(* Logix 5000 project; controller reports 1756-L63 rev 20.11; software revision 20.04; part 52 of 52 *)
(* tags used below, declared in another part *)
   AIT501do : PRANALOG;   // Aeration tank 1 DO
   AIT501ph : PRANALOG;   // Aeration tank 1 pH
   AIT502do : PRANALOG;   // Aeration tank 2 DO
   AIT502ph : PRANALOG;   // Aeration tank 2 pH
   B301 : MOTOR;   // Equalization blower 1
   B302 : MOTOR;   // Equalization blower 2
   B303 : MOTOR;   // Equalization blower 3
   B501 : MOTOR;   // Aeration tank 1 blower 1
   B502 : MOTOR;   // Aeration tank standby blower
   B503 : MOTOR;   // Aeration tank 2 blower 1
   B601 : MOTOR;   // Membrane tank 1 blower
   B602 : MOTOR;   // Membrane tank 2 blower
   B603 : MOTOR;   // Membrane tank 3 blower
   B604 : MOTOR;   // Membrane tank 4 blower
   B901 : MOTOR;   // Digester blower 1
   B902 : MOTOR;   // Digester blower 2
   DIESEL : MOTOR;   // Diesel generator
   FIT201 : PRANALOG;   // Plant influent flow to screens
   FIT701 : PRANALOG;   // Membrane tank 1 permeate flow
   FIT702 : PRANALOG;   // Membrane tank 2 permeate flow
   FIT703 : PRANALOG;   // Membrane tank 3 permeate flow
   FIT704 : PRANALOG;   // Membrane tank 4 permeate flow
   FIT801 : PRANALOG;   // CIP flow
   FIT901 : PRANALOG;   // Membrane tanks 1 & 2 WAS flow
   FIT902 : PRANALOG;   // Membrane tanks 3 & 4 WAS flow
   FunctionBlock_Cycle_Time : REAL;   // Main Task Cycle Time in mseconds
   GT7951 : PRANALOG;   // Screening area H2S monitor
   LIT302 : PRANALOG;   // Equalization tank 302 Level
   LIT501 : PRANALOG;   // Aeration tank 1 Level
   LIT502 : PRANALOG;   // Aeration tank 2 Level
   LIT6101 : PRANALOG;   // Coagulant tank 6101 level
   LIT6102 : PRANALOG;   // Caustic tank 6102 Leve
   P301 : MOTOR;   // Equalization pump 1
   P302 : MOTOR;   // Equalization pump 2
   P303 : MOTOR;   // Equalization pump 3
   P501 : MOTOR;   // Membrane tank 1 mixed liquor pump
   P502 : MOTOR;   // Membrane tank 2 mixed liquor pump
   P503 : MOTOR;   // Membrane tank 3 mixed liquor pump
   P504 : MOTOR;   // Membrane tank 4 mixed liquor pump
   P7011 : MOTOR;   // Membrane tank 1 permeate pump 1
   P7012 : MOTOR;   // Membrane tank 1 permeate pump 2
   P7021 : MOTOR;   // Membrane tank 2 permeate pump 1
   P7022 : MOTOR;   // Membrane tank 2 permeate pump 2
   P7031 : MOTOR;   // Membrane tank 3 permeate pump 1
   P7032 : MOTOR;   // Membrane tank 3 permeate pump 2
   P7041 : MOTOR;   // Membrane tank 4 permeate pump 1
   P7042 : MOTOR;   // Membrane tank 4 permeate pump 2
   P7951 : MOTOR;   // Screen building sump pump
   P801 : MOTOR;   // CIP pump 1
   P802 : MOTOR;   // CIP Pump 2
   P901 : MOTOR;   // Membrane tank 1 WAS pump
   P902 : MOTOR;   // Membrane tank 2 WAS pump
   P903 : MOTOR;   // Digester decant pump
   P904 : MOTOR;   // Membrane tank 4 WAS pump
   P905 : MOTOR;   // Membrane tank 3 WAS pump
   report15_data : LogRecord15[800];
   report15_row_qty : DINT;
   report5_data : LogRecord5[2400];
   report5_row_qty : DINT;
   report_data : LogRecord[200];
   report_pwrup_done : BOOL;
   report_row_daily : DINT;
   SCR201 : MOTOR;   // Inlet screen 1 brush motor
   SCR202 : MOTOR;   // Inlet screen 2 brush motor
   VIT701 : PRANALOG;   // Membrane tank 1 vacuum pressure
   VIT702 : PRANALOG;   // Membrane tank 2 vacuum pressure
   VIT703 : PRANALOG;   // Membrane tank 3 vacuum pressure
   VIT704 : PRANALOG;   // Membrane tank 4 vacuum pressure
   WALLCLOCK : DateTime;   // Global date / time
   WALLCLOCK_lock : BOOL;

PROGRAM MainProgram   (* main routine MainRoutine *)

ROUTINE MainRoutine   (* ladder *)
END_ROUTINE
END_PROGRAM

PROGRAM Report15Calcs   (* main routine Reports *)
VAR
   date_time_current : DateTime := (Year := 2023, Month := 1, Day := 19, Hour := 15, Minute := 26, Second := 14, Microsecond := 9016, DayOfWeek := 4);
   date_time_previous : DateTime := (Year := 2023, Month := 1, Day := 19, Hour := 15, Minute := 26, Second := 14, Microsecond := 9016, DayOfWeek := 4);
   DeleteLog : BOOL;   // Switched on by program to delete logs. Resets when delete is complete
   enable_calc : BOOL := 1;
   ForceDelete : BOOL;   // Switch on to delete contents of log
   max_report_tags : DINT := 20;
   max_tag_idx : DINT := 25;
   MinuteCrt : DINT := 26;
   period_end : BOOL;
   report_row : DINT := 348;
   report_tag_qty : DINT := 20;
   run_val : BOOL;
   tag_idx : DINT;
   tag_valid : BOOL := 1;
   tag_value : REAL := 1.0;
END_VAR

ROUTINE LogCalcRoutine   (* structured text *)
   SBR(tag_value, tag_valid, enable_calc, tag_idx);
   
   (* LogCalc Routine *)
   
   (* Does all processing for log calculations *)
   
   (* Calling parameters: *)
   (*	   tag_value : REAL value of the tag *)
   (*	   tag_valid : BOOL validity of information *)
   (*	   tag_idx : SINT tag index *)
   
   (* Globals used: *)
   
   (* Globals changed: *)
   
   (*-------------------------------------------------------------------------------------------------------------------------------------------------*)
   
   (* check value for quality *)
   tag_value := tag_value;
   (*IF (S:V) THEN
   	tag_value := 0;
   	tag_valid := 0;
   	enable_calc := 0;
   END_IF;*)
   
   (* only calculate if it is enabled *)
   IF enable_calc THEN
   	(* check for valid data *)
   	IF  NOT (tag_value = tag_value) THEN
   		tag_valid := 0;
   		tag_value := 0;
   	END_IF;
   
   	(* calculate the max and min *)
   
   	(* if this is the first time this hour, set max and min to current value *)
   	IF report15_data[report_row].log_data[tag_idx].time = 0 THEN
   		report15_data[report_row].log_data[tag_idx].max := tag_value;
   		report15_data[report_row].log_data[tag_idx].min := tag_value;
   		report15_data[report_row].log_data[tag_idx].maxminute := MinuteCrt;
   		report15_data[report_row].log_data[tag_idx].minminute := MinuteCrt;
   
   	(* otherwise, check to see if max or min has been exceeded *)
   	ELSE
   		IF tag_value > report15_data[report_row].log_data[tag_idx].max THEN
   		    report15_data[report_row].log_data[tag_idx].max := tag_value;
   			report15_data[report_row].log_data[tag_idx].maxminute := MinuteCrt;
   		ELSIF tag_value < report15_data[report_row].log_data[tag_idx].min THEN
   		    report15_data[report_row].log_data[tag_idx].min := tag_value;
   			report15_data[report_row].log_data[tag_idx].minminute := MinuteCrt;
   		END_IF;
   	END_IF;
   
   
   	(* add to the total *)
   	report15_data[report_row].log_data[tag_idx].total := report15_data[report_row].log_data[tag_idx].total + FunctionBlock_Cycle_Time / 1000 * tag_value;
   
   	(* add to the time *)
   	report15_data[report_row].log_data[tag_idx].time := report15_data[report_row].log_data[tag_idx].time + FunctionBlock_Cycle_Time / 1000;
   
   	(* Valid *)
   	IF NOT (tag_valid) THEN
   		report15_data[report_row].log_data[tag_idx].valid := 0;
   	END_IF;
   
   END_IF;
END_ROUTINE

ROUTINE LogDeleteRoutine   (* structured text *)
// Deletes log and resets it to Zero
   SBR();
   
   (* LogDelete Routine *)
   
   (* Does all processing to clear out Log *)
   
   (* Calling parameters: *)
   
   (* Globals used: *)
   
   (* Globals changed: *)
   
   (*-------------------------------------------------------------------------------------------------------------------------------------------------*)
   
   
   (* set the timestamp for the finished row *)
   report15_data[report_row].time.Year := 0;
   report15_data[report_row].time.Month := 0;
   report15_data[report_row].time.Day := 0;
   report15_data[report_row].time.Hour := 0;
   report15_data[report_row].time.Minute := 0;
   report15_data[report_row].time.Second := 0;
   report15_data[report_row].time.DST_ON := 0;
   
   (* Go to next record *)
   report_row := report_row + 1;
   IF report_row >= report15_row_qty THEN
   	report_row := 0;
   END_IF;
   
   (* clear the timestamp for the new row *)
   report15_data[report_row].time.Year := 0;
   report15_data[report_row].time.Month := 0;
   report15_data[report_row].time.Day := 0;
   report15_data[report_row].time.Hour := 0;
   report15_data[report_row].time.Minute := 0;
   report15_data[report_row].time.Second := 0;
   report15_data[report_row].time.DST_ON := 0;
   
   (* Do initialisation for the new record *)
   FOR tag_idx := 0 to report_tag_qty - 1 DO
   	report15_data[report_row].log_data[tag_idx].min := 0;
   	report15_data[report_row].log_data[tag_idx].max := 0;
   	report15_data[report_row].log_data[tag_idx].total := 0;
   	report15_data[report_row].log_data[tag_idx].time := 0;
   	report15_data[report_row].log_data[tag_idx].valid := 1;
   END_FOR;
   
   (* Do initialisation for the new record *)
   SIZE(report15_data[report_row].log_data[0],0,max_report_tags);
   max_report_tags := report_tag_qty;  // to be deleted if above line is correct  this will allow clearing of the full table
   FOR tag_idx := 0 to max_report_tags - 1 DO
   	report15_data[report_row].log_data[tag_idx].min := 0;
   	report15_data[report_row].log_data[tag_idx].max := 0;
   	report15_data[report_row].log_data[tag_idx].total := 0;
   	report15_data[report_row].log_data[tag_idx].time := 0;
   	report15_data[report_row].log_data[tag_idx].minminute := 0;
   	report15_data[report_row].log_data[tag_idx].maxminute := 0;
   	report15_data[report_row].log_data[tag_idx].valid := 1;
   END_FOR;
   
   (* If this is the last row to delete (i.e. row 0) end the delete *)
   IF report_row = 0 THEN
   	DeleteLog := 0;
   END_IF;
END_ROUTINE

ROUTINE LogMotorRoutine   (* structured text *)
   SBR(run_val, tag_idx);
   
   IF run_val THEN
   	JSR(LogCalcRoutine, 4 , 1.0, 1, 1, tag_idx);
   ELSE
   	JSR(LogCalcRoutine, 4 , 0.0, 1, 1, tag_idx);
   END_IF;
   
END_ROUTINE

ROUTINE LogSaveRoutine   (* structured text *)
   SBR();
   
   (* LogSave Routine *)
   
   (* Does all processing for saving log data at the end of the hour *)
   
   (* Calling parameters: *)
   
   (* Globals used: *)
   
   (* Globals changed: *)
   
   (*-------------------------------------------------------------------------------------------------------------------------------------------------*)
   
   
   (* set the timestamp for the finished row *)
   report15_data[report_row].time.Year := date_time_previous.Year;
   report15_data[report_row].time.Month := date_time_previous.Month;
   report15_data[report_row].time.Day := date_time_previous.Day;
   report15_data[report_row].time.Hour := date_time_previous.Hour;
   report15_data[report_row].time.Minute := date_time_previous.Minute;
   report15_data[report_row].time.Second := date_time_previous.Second;
   report15_data[report_row].time.DST_ON := date_time_previous.DST_ON;
   
   (* Go to next record *)
   report_row := report_row + 1;
   IF report_row >= report15_row_qty THEN
   	report_row := 0;
   END_IF;
   
   (* clear the timestamp for the new row *)
   report15_data[report_row].time.Year := 0;
   report15_data[report_row].time.Month := 0;
   report15_data[report_row].time.Day := 0;
   report15_data[report_row].time.Hour := 0;
   report15_data[report_row].time.Minute := 0;
   report15_data[report_row].time.Second := 0;
   report15_data[report_row].time.DST_ON := 0;
   
   (* Do initialisation for the new record *)
   FOR tag_idx := 0 to report_tag_qty - 1 DO
   	report15_data[report_row].log_data[tag_idx].min := 0;
   	report15_data[report_row].log_data[tag_idx].max := 0;
   	report15_data[report_row].log_data[tag_idx].total := 0;
   	report15_data[report_row].log_data[tag_idx].time := 0;
   	report15_data[report_row].log_data[tag_idx].valid := 1;
   END_FOR;
   
   (* Do initialisation for the new record *)
   SIZE(report15_data[report_row].log_data[0],0,max_report_tags);
   max_report_tags := report_tag_qty;  // to be deleted if above line is correct  this will allow clearing of the full table
   FOR tag_idx := 0 to max_report_tags - 1 DO
   	report15_data[report_row].log_data[tag_idx].min := 0;
   	report15_data[report_row].log_data[tag_idx].max := 0;
   	report15_data[report_row].log_data[tag_idx].total := 0;
   	report15_data[report_row].log_data[tag_idx].time := 0;
   	report15_data[report_row].log_data[tag_idx].minminute := 0;
   	report15_data[report_row].log_data[tag_idx].maxminute := 0;
   	report15_data[report_row].log_data[tag_idx].valid := 1;
   END_FOR;
END_ROUTINE

ROUTINE Reports   (* structured text *)
   (* Report logging processing program *)
   
   (* Does all processing for logging of report data *)
   
   (* Globals used: *)
   
   (* Globals changed: *)
   
   (*-------------------------------------------------------------------------------------------------------------------------------------------------*)
   
   
   //**********************to be adjusted by programmer ********************************
   SIZE(report15_data[0],0,report15_row_qty);
   SIZE(report15_data[0].log_data[0],0,report_tag_qty);
   //***********************************************************************************
   
   (* Get current date/time *)
   IF NOT WALLCLOCK_lock THEN
   	cop( WALLCLOCK, date_time_current, 1);
   END_IF;
   
   (* adjust previous hour if dst changed *)
   IF date_time_current.DST_ON AND NOT date_time_previous.DST_ON THEN
   	date_time_previous.Hour := date_time_previous.Hour + 1;
   ELSIF NOT date_time_current.DST_ON AND date_time_previous.DST_ON THEN
   	date_time_previous.Hour := date_time_previous.Hour - 1;
   END_IF;
   
   (* Detect 15 minute change to see if the period is over *)
   IF date_time_current.Minute <> date_time_previous.Minute THEN
   	period_end := (date_time_current.Minute / 15) <> (date_time_previous.Minute / 15);
   ELSE
   	period_end := 0;
   END_IF;
   
   (* if the hour just ended, save the new hour's data *)
   IF period_end THEN
   	JSR(LogSaveRoutine);
   END_IF;
   
   (* delete log logic, used to clear out data log *)
   If ForceDelete AND NOT DeleteLog THEN
   	DeleteLog := 1;
   	report_row := 1;
   END_IF;
   If DeleteLog THEN
   	JSR(LogDeleteRoutine);
   END_IF;
   ForceDelete := 0;
   
   MinuteCrt := date_time_current.Minute;
   
   
   // Keep track of time reported, enabled in routine with most frequent active data collection
   JSR( LogCalcRoutine, 4, 1.0, 1, 1, 0);  //duration
   
   
   (************ insert logs here ***************)
   
   
   
   
   (* keep track of the last date for the end of the hour *)
   COP(date_time_current,date_time_previous,1);
   
END_ROUTINE
END_PROGRAM

PROGRAM Report5Calcs   (* main routine Reports *)
VAR
   date_time_current : DateTime := (Year := 2023, Month := 1, Day := 19, Hour := 15, Minute := 26, Second := 14, Microsecond := 9016, DayOfWeek := 4);
   date_time_previous : DateTime := (Year := 2023, Month := 1, Day := 19, Hour := 15, Minute := 26, Second := 14, Microsecond := 9016, DayOfWeek := 4);
   DeleteLog : BOOL;   // Switched on by program to delete logs. Resets when delete is complete
   enable_calc : BOOL := 1;
   ForceDelete : BOOL;   // Switch on to delete contents of log
   max_report_tags : DINT := 20;
   max_tag_idx : DINT := 25;
   MinuteCrt : DINT := 26;
   period_end : BOOL;
   report_row : DINT := 469;
   report_tag_qty : DINT := 20;
   run_val : BOOL;
   tag_idx : DINT;
   tag_valid : BOOL := 1;
   tag_value : REAL := 1.0;
END_VAR

ROUTINE LogCalcRoutine   (* structured text *)
   SBR(tag_value, tag_valid, enable_calc, tag_idx);
   
   (* LogCalc Routine *)
   
   (* Does all processing for log calculations *)
   
   (* Calling parameters: *)
   (*	   tag_value : REAL value of the tag *)
   (*	   tag_valid : BOOL validity of information *)
   (*	   tag_idx : SINT tag index *)
   
   (* Globals used: *)
   
   (* Globals changed: *)
   
   (*-------------------------------------------------------------------------------------------------------------------------------------------------*)
   
   (* check value for quality *)
   tag_value := tag_value;
   (*IF (S:V) THEN
   	tag_value := 0;
   	tag_valid := 0;
   	enable_calc := 0;
   END_IF;*)
   
   (* only calculate if it is enabled *)
   IF enable_calc THEN
   	(* check for valid data *)
   	IF  NOT (tag_value = tag_value) THEN
   		tag_valid := 0;
   		tag_value := 0;
   	END_IF;
   
   	(* calculate the max and min *)
   
   	(* if this is the first time this hour, set max and min to current value *)
   	IF report5_data[report_row].log_data[tag_idx].time = 0 THEN
   		report5_data[report_row].log_data[tag_idx].max := tag_value;
   		report5_data[report_row].log_data[tag_idx].min := tag_value;
   		report5_data[report_row].log_data[tag_idx].maxminute := MinuteCrt;
   		report5_data[report_row].log_data[tag_idx].minminute := MinuteCrt;
   
   	(* otherwise, check to see if max or min has been exceeded *)
   	ELSE
   		IF tag_value > report5_data[report_row].log_data[tag_idx].max THEN
   		    report5_data[report_row].log_data[tag_idx].max := tag_value;
   			report5_data[report_row].log_data[tag_idx].maxminute := MinuteCrt;
   		ELSIF tag_value < report5_data[report_row].log_data[tag_idx].min THEN
   		    report5_data[report_row].log_data[tag_idx].min := tag_value;
   			report5_data[report_row].log_data[tag_idx].minminute := MinuteCrt;
   		END_IF;
   	END_IF;
   
   
   	(* add to the total *)
   	report5_data[report_row].log_data[tag_idx].total := report5_data[report_row].log_data[tag_idx].total + FunctionBlock_Cycle_Time / 1000 * tag_value;
   
   	(* add to the time *)
   	report5_data[report_row].log_data[tag_idx].time := report5_data[report_row].log_data[tag_idx].time + FunctionBlock_Cycle_Time / 1000;
   
   	(* Valid *)
   	IF NOT (tag_valid) THEN
   		report5_data[report_row].log_data[tag_idx].valid := 0;
   	END_IF;
   
   END_IF;
END_ROUTINE

ROUTINE LogDeleteRoutine   (* structured text *)
// Deletes log and resets it to Zero
   SBR();
   
   (* LogDelete Routine *)
   
   (* Does all processing to clear out Log *)
   
   (* Calling parameters: *)
   
   (* Globals used: *)
   
   (* Globals changed: *)
   
   (*-------------------------------------------------------------------------------------------------------------------------------------------------*)
   
   
   (* set the timestamp for the finished row *)
   report5_data[report_row].time.Year := 0;
   report5_data[report_row].time.Month := 0;
   report5_data[report_row].time.Day := 0;
   report5_data[report_row].time.Hour := 0;
   report5_data[report_row].time.Minute := 0;
   report5_data[report_row].time.Second := 0;
   report5_data[report_row].time.DST_ON := 0;
   
   (* Go to next record *)
   report_row := report_row + 1;
   IF report_row >= report5_row_qty THEN
   	report_row := 0;
   END_IF;
   
   (* clear the timestamp for the new row *)
   report5_data[report_row].time.Year := 0;
   report5_data[report_row].time.Month := 0;
   report5_data[report_row].time.Day := 0;
   report5_data[report_row].time.Hour := 0;
   report5_data[report_row].time.Minute := 0;
   report5_data[report_row].time.Second := 0;
   report5_data[report_row].time.DST_ON := 0;
   
   (* Do initialisation for the new record *)
   FOR tag_idx := 0 to report_tag_qty - 1 DO
   	report5_data[report_row].log_data[tag_idx].min := 0;
   	report5_data[report_row].log_data[tag_idx].max := 0;
   	report5_data[report_row].log_data[tag_idx].total := 0;
   	report5_data[report_row].log_data[tag_idx].time := 0;
   	report5_data[report_row].log_data[tag_idx].valid := 1;
   END_FOR;
   
   (* Do initialisation for the new record *)
   SIZE(report5_data[report_row].log_data[0],0,max_report_tags);
   max_report_tags := report_tag_qty;  // to be deleted if above line is correct  this will allow clearing of the full table
   FOR tag_idx := 0 to max_report_tags - 1 DO
   	report5_data[report_row].log_data[tag_idx].min := 0;
   	report5_data[report_row].log_data[tag_idx].max := 0;
   	report5_data[report_row].log_data[tag_idx].total := 0;
   	report5_data[report_row].log_data[tag_idx].time := 0;
   	report5_data[report_row].log_data[tag_idx].minminute := 0;
   	report5_data[report_row].log_data[tag_idx].maxminute := 0;
   	report5_data[report_row].log_data[tag_idx].valid := 1;
   END_FOR;
   
   (* If this is the last row to delete (i.e. row 0) end the delete *)
   IF report_row = 0 THEN
   	DeleteLog := 0;
   END_IF;
END_ROUTINE

ROUTINE LogMotorRoutine   (* structured text *)
   SBR(run_val, tag_idx);
   
   IF run_val THEN
   	JSR(LogCalcRoutine, 4 , 1.0, 1, 1, tag_idx);
   ELSE
   	JSR(LogCalcRoutine, 4 , 0.0, 1, 1, tag_idx);
   END_IF;
   
END_ROUTINE

ROUTINE LogSaveRoutine   (* structured text *)
   SBR();
   
   (* LogSave Routine *)
   
   (* Does all processing for saving log data at the end of the hour *)
   
   (* Calling parameters: *)
   
   (* Globals used: *)
   
   (* Globals changed: *)
   
   (*-------------------------------------------------------------------------------------------------------------------------------------------------*)
   
   
   (* set the timestamp for the finished row *)
   report5_data[report_row].time.Year := date_time_previous.Year;
   report5_data[report_row].time.Month := date_time_previous.Month;
   report5_data[report_row].time.Day := date_time_previous.Day;
   report5_data[report_row].time.Hour := date_time_previous.Hour;
   report5_data[report_row].time.Minute := date_time_previous.Minute;
   report5_data[report_row].time.Second := date_time_previous.Second;
   report5_data[report_row].time.DST_ON := date_time_previous.DST_ON;
   
   (* Go to next record *)
   report_row := report_row + 1;
   IF report_row >= report5_row_qty THEN
   	report_row := 0;
   END_IF;
   
   (* clear the timestamp for the new row *)
   report5_data[report_row].time.Year := 0;
   report5_data[report_row].time.Month := 0;
   report5_data[report_row].time.Day := 0;
   report5_data[report_row].time.Hour := 0;
   report5_data[report_row].time.Minute := 0;
   report5_data[report_row].time.Second := 0;
   report5_data[report_row].time.DST_ON := 0;
   
   (* Do initialisation for the new record *)
   FOR tag_idx := 0 to report_tag_qty - 1 DO
   	report5_data[report_row].log_data[tag_idx].min := 0;
   	report5_data[report_row].log_data[tag_idx].max := 0;
   	report5_data[report_row].log_data[tag_idx].total := 0;
   	report5_data[report_row].log_data[tag_idx].time := 0;
   	report5_data[report_row].log_data[tag_idx].valid := 1;
   END_FOR;
   
   (* Do initialisation for the new record *)
   SIZE(report5_data[report_row].log_data[0],0,max_report_tags);
   max_report_tags := report_tag_qty;  // to be deleted if above line is correct  this will allow clearing of the full table
   FOR tag_idx := 0 to max_report_tags - 1 DO
   	report5_data[report_row].log_data[tag_idx].min := 0;
   	report5_data[report_row].log_data[tag_idx].max := 0;
   	report5_data[report_row].log_data[tag_idx].total := 0;
   	report5_data[report_row].log_data[tag_idx].time := 0;
   	report5_data[report_row].log_data[tag_idx].minminute := 0;
   	report5_data[report_row].log_data[tag_idx].maxminute := 0;
   	report5_data[report_row].log_data[tag_idx].valid := 1;
   END_FOR;
END_ROUTINE

ROUTINE Reports   (* structured text *)
   (* Report logging processing program *)
   
   (* Does all processing for logging of report data *)
   
   (* Globals used: *)
   
   (* Globals changed: *)
   
   (*-------------------------------------------------------------------------------------------------------------------------------------------------*)
   
   
   //**********************to be adjusted by programmer ********************************
   SIZE(report5_data[0],0,report5_row_qty);
   SIZE(report5_data[0].log_data[0],0,report_tag_qty);
   
   //***********************************************************************************
   
   (* Get current date/time *)
   IF NOT WALLCLOCK_lock THEN
   	cop( WALLCLOCK, date_time_current, 1);
   END_IF;
   
   (* adjust previous hour if dst changed *)
   IF date_time_current.DST_ON AND NOT date_time_previous.DST_ON THEN
   	date_time_previous.Hour := date_time_previous.Hour + 1;
   ELSIF NOT date_time_current.DST_ON AND date_time_previous.DST_ON THEN
   	date_time_previous.Hour := date_time_previous.Hour - 1;
   END_IF;
   
   (* Detect 5 minute change to see if the period is over *)
   IF date_time_current.Minute <> date_time_previous.Minute THEN
   	period_end := (date_time_current.Minute / 5) <> (date_time_previous.Minute / 5);
   ELSE
   	period_end := 0;
   END_IF;
   
   (* if the hour just ended, save the new hour's data *)
   IF period_end THEN
   	JSR(LogSaveRoutine);
   END_IF;
   
   (* delete log logic, used to clear out data log *)
   If ForceDelete AND NOT DeleteLog THEN
   	DeleteLog := 1;
   	report_row := 1;
   END_IF;
   If DeleteLog THEN
   	JSR(LogDeleteRoutine);
   END_IF;
   ForceDelete := 0;
   
   
   MinuteCrt := date_time_current.Minute;
   
   // Keep track of time reported, enabled in routine with most frequent active data collection
   JSR( LogCalcRoutine, 4, 1.0, 1, 1, 0);  //duration
   
   
   
   (************ insert logs here ***************)
   
   
   
   
   (* keep track of the last date for the end of the hour *)
   COP(date_time_current,date_time_previous,1);
   
END_ROUTINE
END_PROGRAM

PROGRAM ReportCalcs   (* main routine Reports *)
VAR
   date_time_current : DateTime := (Year := 2023, Month := 1, Day := 19, Hour := 15, Minute := 26, Second := 14, Microsecond := 9016, DayOfWeek := 4);
   date_time_previous : DateTime := (Year := 2023, Month := 1, Day := 19, Hour := 15, Minute := 26, Second := 14, Microsecond := 9016, DayOfWeek := 4);
   DeleteLog : BOOL;   // Switched on by program to delete logs. Resets when delete is complete
   enable_calc : BOOL := 1;
   ForceDelete : BOOL;   // Switch on to delete contents of log
   hour_end : BOOL;
   max_report_tags : DINT := 125;
   max_tag_idx : DINT := 25;
   MinuteCrt : DINT := 26;
   POOP : BOOL;
   report_row : DINT := 156;
   run_val : BOOL;
   tag_idx : DINT := 60;
   tag_valid : BOOL := 1;
   tag_value : REAL;
END_VAR

ROUTINE LogCalcRoutine   (* structured text *)
   SBR(tag_value, tag_valid, enable_calc, tag_idx);
   
   (* LogCalc Routine *)
   
   (* Does all processing for log calculations *)
   
   (* Calling parameters: *)
   (*	   tag_value : REAL value of the tag *)
   (*	   tag_valid : BOOL validity of information *)
   (*	   tag_idx : SINT tag index *)
   
   (* Globals used: *)
   
   (* Globals changed: *)
   
   (*-------------------------------------------------------------------------------------------------------------------------------------------------*)
   
   (* check value for quality *)
   tag_value := tag_value;
   (*IF (S:V) THEN
   	tag_value := 0;
   	tag_valid := 0;
   	enable_calc := 0;
   END_IF;*)
   
   (* only calculate if it is enabled *)
   IF enable_calc THEN
   	(* check for valid data *)
   	IF  NOT (tag_value = tag_value) THEN
   		tag_valid := 0;
   		tag_value := 0;
   	END_IF;
   
   	(* calculate the max and min *)
   
   	(* if this is the first time this hour, set max and min to current value *)
   	IF report_data[report_row].log_data[tag_idx].time = 0 THEN
   		report_data[report_row].log_data[tag_idx].max := tag_value;
   		report_data[report_row].log_data[tag_idx].min := tag_value;
   		report_data[report_row].log_data[tag_idx].maxminute := MinuteCrt;
   		report_data[report_row].log_data[tag_idx].minminute := MinuteCrt;
   
   	(* otherwise, check to see if max or min has been exceeded *)
   	ELSE
   		IF tag_value > report_data[report_row].log_data[tag_idx].max THEN
   		    report_data[report_row].log_data[tag_idx].max := tag_value;
   			report_data[report_row].log_data[tag_idx].maxminute := MinuteCrt;
   		ELSIF tag_value < report_data[report_row].log_data[tag_idx].min THEN
   		    report_data[report_row].log_data[tag_idx].min := tag_value;
   			report_data[report_row].log_data[tag_idx].minminute := MinuteCrt;
   		END_IF;
   	END_IF;
   
   
   	(* add to the total *)
   	report_data[report_row].log_data[tag_idx].total := report_data[report_row].log_data[tag_idx].total + FunctionBlock_Cycle_Time / 1000 * tag_value;
   
   	(* add to the time *)
   	report_data[report_row].log_data[tag_idx].time := report_data[report_row].log_data[tag_idx].time + FunctionBlock_Cycle_Time / 1000;
   
   	(* Valid *)
   	IF NOT (tag_valid) THEN
   		report_data[report_row].log_data[tag_idx].valid := 0;
   	END_IF;
   
   END_IF;
END_ROUTINE

ROUTINE LogDeleteRoutine   (* structured text *)
// Deletes log and resets it to Zero
   SBR();
   
   (* LogDelete Routine *)
   
   (* Does all processing to clear out Log *)
   
   (* Calling parameters: *)
   
   (* Globals used: *)
   
   (* Globals changed: *)
   
   (*-------------------------------------------------------------------------------------------------------------------------------------------------*)
   
   FOR report_row := 0 TO report_row_qty - 1 DO
   
   	(* clear the timestamp  *)
   	report_data[report_row].time.Year := 0;
   	report_data[report_row].time.Month := 0;
   	report_data[report_row].time.Day := 0;
   	report_data[report_row].time.Hour := 0;
   	report_data[report_row].time.Minute := 0;
   	report_data[report_row].time.Second := 0;
   	report_data[report_row].time.DST_ON := 0;
   
   	FOR tag_idx := 0 to report_tag_qty - 1 DO
   		report_data[report_row].log_data[tag_idx].min := 0;
   		report_data[report_row].log_data[tag_idx].max := 0;
   		report_data[report_row].log_data[tag_idx].total := 0;
   		report_data[report_row].log_data[tag_idx].time := 0;
   		report_data[report_row].log_data[tag_idx].valid := 1;
   	END_FOR;
   
   END_FOR;
   
   
   (* Set the current row to 0 and end the delete *)
   report_row := 0;
   DeleteLog := 0;
   
END_ROUTINE

ROUTINE LogMotorRoutine   (* structured text *)
   SBR(run_val, tag_idx);
   
   IF run_val THEN
   	JSR(LogCalcRoutine, 4 , 1.0, 1, 1, tag_idx);
   ELSE
   	JSR(LogCalcRoutine, 4 , 0.0, 1, 1, tag_idx);
   END_IF;
   
END_ROUTINE

ROUTINE LogSaveRoutine   (* structured text *)
   SBR();
   
   (* LogSave Routine *)
   
   (* Does all processing for saving log data at the end of the hour *)
   
   (* Calling parameters: *)
   
   (* Globals used: *)
   
   (* Globals changed: *)
   
   (*-------------------------------------------------------------------------------------------------------------------------------------------------*)
   
   
   (* set the timestamp for the finished row *)
   report_data[report_row].time.Year := date_time_previous.Year;
   report_data[report_row].time.Month := date_time_previous.Month;
   report_data[report_row].time.Day := date_time_previous.Day;
   report_data[report_row].time.Hour := date_time_previous.Hour;
   report_data[report_row].time.Minute := date_time_previous.Minute;
   report_data[report_row].time.Second := date_time_previous.Second;
   report_data[report_row].time.DST_ON := date_time_previous.DST_ON;
   
   (* Go to next record *)
   report_row := report_row + 1;
   IF report_row >= report_row_qty THEN
   	report_row := 0;
   END_IF;
   
   (* clear the timestamp for the new row *)
   report_data[report_row].time.Year := 0;
   report_data[report_row].time.Month := 0;
   report_data[report_row].time.Day := 0;
   report_data[report_row].time.Hour := 0;
   report_data[report_row].time.Minute := 0;
   report_data[report_row].time.Second := 0;
   report_data[report_row].time.DST_ON := 0;
   
   (* Do initialisation for the new record *)
   FOR tag_idx := 0 to report_tag_qty - 1 DO
   	report_data[report_row].log_data[tag_idx].min := 0;
   	report_data[report_row].log_data[tag_idx].max := 0;
   	report_data[report_row].log_data[tag_idx].total := 0;
   	report_data[report_row].log_data[tag_idx].time := 0;
   	report_data[report_row].log_data[tag_idx].valid := 1;
   END_FOR;
   
   (* Do initialisation for the new record *)
   SIZE(report_data[report_row].log_data[0],0,max_report_tags);
   max_report_tags := report_tag_qty;  // to be deleted if above line is correct  this will allow clearing of the full table
   FOR tag_idx := 0 to max_report_tags - 1 DO
   	report_data[report_row].log_data[tag_idx].min := 0;
   	report_data[report_row].log_data[tag_idx].max := 0;
   	report_data[report_row].log_data[tag_idx].total := 0;
   	report_data[report_row].log_data[tag_idx].time := 0;
   	report_data[report_row].log_data[tag_idx].minminute := 0;
   	report_data[report_row].log_data[tag_idx].maxminute := 0;
   	report_data[report_row].log_data[tag_idx].valid := 1;
   END_FOR;
END_ROUTINE

ROUTINE Reports   (* structured text *)
   (* Report logging processing program *)
   
   (* Does all processing for logging of report data *)
   
   (* Globals used: *)
   
   (* Globals changed: *)
   
   (*-------------------------------------------------------------------------------------------------------------------------------------------------*)
   
   
   //**********************to be adjusted by programmer ********************************
   SIZE(report_data[0].log_data[0],0,report_tag_qty);
   SIZE(report_data[0],0,report_row_qty);
   //***********************************************************************************
   
   (* Get current date/time *)
   IF NOT WALLCLOCK_lock THEN
   	cop( WALLCLOCK, date_time_current, 1);
   END_IF;
   
   (* adjust previous hour if dst changed *)
   IF date_time_current.DST_ON AND NOT date_time_previous.DST_ON THEN
   	date_time_previous.Hour := date_time_previous.Hour + 1;
   ELSIF NOT date_time_current.DST_ON AND date_time_previous.DST_ON THEN
   	date_time_previous.Hour := date_time_previous.Hour - 1;
   END_IF;
   
   (* Detect hour change to see if the period is over *)
   IF date_time_current.Hour <> date_time_previous.Hour THEN
   	hour_end := 1;
   ELSE
   	hour_end := 0;
   END_IF;
   
   (* if the hour just ended, save the new hour's data *)
   IF hour_end OR POOP THEN
   	JSR(LogSaveRoutine);
   END_IF;
   POOP := 0;
   
   (* delete log logic, used to clear out data log *)
   If ForceDelete AND NOT DeleteLog THEN
   	DeleteLog := 1;
   END_IF;
   If DeleteLog THEN
   	JSR(LogDeleteRoutine);
   END_IF;
   ForceDelete := 0;
   
   MinuteCrt := date_time_current.Minute;
   
   // Keep track of time reported, enabled in routine with most frequent active data collection
   JSR( LogCalcRoutine, 4, 1.0, 1, 1, 0);  //duration
   
   (************ insert logs here ***************)
   
   JSR( LogMotorRoutine, 2, SCR201.run_sts, 1 );  //SCR201 - Inlet screen 1 brush motor
   JSR( LogMotorRoutine, 2, SCR202.run_sts, 2 );  //SCR202 - Inlet screen 2 brush motor
   JSR( LogMotorRoutine, 2, P301.run_sts, 3 );  //P301 - Equalization pump 1
   JSR( LogMotorRoutine, 2, P302.run_sts, 4 );  //P302 - Equalization pump 2
   JSR( LogMotorRoutine, 2, P303.run_sts, 5 );  //P303 - Equalization pump 3
   JSR( LogMotorRoutine, 2, P501.run_sts, 6 );  //P501 - Membrane tank 1 mixed liquor pump
   JSR( LogMotorRoutine, 2, P502.run_sts, 7 );  //P502 - Membrane tank 2 mixed liquor pump
   JSR( LogMotorRoutine, 2, P503.run_sts, 8 );  //P503 - Membrane tank 3 mixed liquor pump
   JSR( LogMotorRoutine, 2, P504.run_sts, 9 );  //P504 - Membrane tank 4 mixed liquor pump
   JSR( LogMotorRoutine, 2, P903.run_sts, 10 );  //P903 - Digester decant pump
   JSR( LogMotorRoutine, 2, DIESEL.run_sts, 11 );  //DIESEL - Diesel generator
   JSR( LogMotorRoutine, 2, B301.run_sts, 12 );  //B301 - Equalization blower 1
   JSR( LogMotorRoutine, 2, B302.run_sts, 13 );  //B302 - Equalization blower 2
   JSR( LogMotorRoutine, 2, B303.run_sts, 14 );  //B303 - Equalization blower 3
   JSR( LogMotorRoutine, 2, B501.run_sts, 15 );  //B501 - Aeration tank 1 blower 1
   JSR( LogMotorRoutine, 2, B502.run_sts, 16 );  //B502 - Aeration tank standby blower
   JSR( LogMotorRoutine, 2, B503.run_sts, 17 );  //B503 - Aeration tank 2 blower 1
   JSR( LogMotorRoutine, 2, B601.run_sts, 18 );  //B601 - Membrane tank 1 blower
   JSR( LogMotorRoutine, 2, B602.run_sts, 19 );  //B602 - Membrane tank 2 blower
   JSR( LogMotorRoutine, 2, B901.run_sts, 20 );  //B901 - Digester blower 1
   JSR( LogMotorRoutine, 2, B902.run_sts, 21 );  //B902 - Digester blower 2
   JSR( LogMotorRoutine, 2, P901.run_sts, 22 );  //P901 - Membrane tank 1 WAS pump
   JSR( LogMotorRoutine, 2, P7011.run_sts, 23 );  //P7011 - Membrane tank 1 permeate pump 1
   JSR( LogMotorRoutine, 2, P7012.run_sts, 24 );  //P7012 - Membrane tank 1 permeate pump 2
   JSR( LogMotorRoutine, 2, P902.run_sts, 25 );  //P902 - Membrane tank 2 WAS pump
   JSR( LogMotorRoutine, 2, P7021.run_sts, 26 );  //P7021 - Membrane tank 2 permeate pump 1
   JSR( LogMotorRoutine, 2, P7022.run_sts, 27 );  //P7022 - Membrane tank 2 permeate pump 2
   JSR( LogMotorRoutine, 2, P801.run_sts, 28 );  //P801 - CIP pump
   JSR( LogMotorRoutine, 2, B603.run_sts, 29 );  //B603 - Membrane tank 3 blower
   JSR( LogMotorRoutine, 2, B604.run_sts, 30 );  //B604 - Membrane tank 4 blower
   JSR( LogMotorRoutine, 2, P7031.run_sts, 31 );  //P7031 - Membrane tank 3 permeate pump 1
   JSR( LogMotorRoutine, 2, P7032.run_sts, 32 );  //P7032 - Membrane tank 3 permeate pump 2
   JSR( LogMotorRoutine, 2, P905.run_sts, 33 );  //P905 - Membrane tank 3 WAS pump
   JSR( LogMotorRoutine, 2, P904.run_sts, 34 );  //P904 - Membrane tank 4 WAS pump
   JSR( LogMotorRoutine, 2, P7041.run_sts, 35 );  //P7041 - Membrane tank 4 permeate pump 1
   JSR( LogMotorRoutine, 2, P7042.run_sts, 36 );  //P7042 - Membrane tank 4 permeate pump 2
   JSR( LogCalcRoutine, 4, FIT201.value, FIT201.valid, FIT201.log, 37);  //FIT201 - Plant influent flow to screens
   JSR( LogCalcRoutine, 4, GT7951.value, GT7951.valid, GT7951.log, 38);  //GT7951 - Screening area H2S monitor
   JSR( LogCalcRoutine, 4, LIT302.value, LIT302.valid, LIT302.log, 39);  //LIT302 - Equalization tank 302 Level
   JSR( LogCalcRoutine, 4, AIT501ph.value, AIT501ph.valid, AIT501ph.log, 40);  //AIT501ph - Aeration tank 1 pH
   JSR( LogCalcRoutine, 4, AIT501do.value, AIT501do.valid, AIT501do.log, 41);  //AIT501do - Aeration tank 1 DO
   JSR( LogCalcRoutine, 4, LIT501.value, LIT501.valid, LIT501.log, 42);  //LIT501 - Aeration tank 1 Level
   JSR( LogCalcRoutine, 4, VIT701.value, VIT701.valid, VIT701.log, 43);  //VIT701 - Membrane tank 1 vacuum pressure
   JSR( LogCalcRoutine, 4, VIT702.value, VIT702.valid, VIT702.log, 44);  //VIT702 - Membrane tank 2 vacuum pressure
   JSR( LogCalcRoutine, 4, FIT701.value, FIT701.valid, FIT701.log, 45);  //FIT701 - Membrane tank 1 permeate flow
   JSR( LogCalcRoutine, 4, FIT702.value, FIT702.valid, FIT702.log, 46);  //FIT702 - Membrane tank 2 permeate flow
   JSR( LogCalcRoutine, 4, FIT901.value, FIT901.valid, FIT901.log, 47);  //FIT901 - Membrane tanks 1 & 2 WAS flow
   JSR( LogCalcRoutine, 4, AIT502ph.value, AIT502ph.valid, AIT502ph.log, 48);  //AIT502ph - Aeration tank 2 pH
   JSR( LogCalcRoutine, 4, AIT502do.value, AIT502do.valid, AIT502do.log, 49);  //AIT502do - Aeration tank 2 DO
   JSR( LogCalcRoutine, 4, LIT502.value, LIT502.valid, LIT502.log, 50);  //LIT502 - Aeration tank 2 Level
   JSR( LogCalcRoutine, 4, FIT902.value, FIT902.valid, FIT902.log, 51);  //FIT902 - Membrane tanks 3 & 4 WAS flow
   JSR( LogCalcRoutine, 4, VIT703.value, VIT703.valid, VIT703.log, 52);  //VIT703 - Membrane tank 3 vacuum pressure
   JSR( LogCalcRoutine, 4, VIT704.value, VIT704.valid, VIT704.log, 53);  //VIT704 - Membrane tank 4 vacuum pressure
   JSR( LogCalcRoutine, 4, FIT703.value, FIT703.valid, FIT703.log, 54);  //FIT703 - Membrane tank 3 permeate flow
   JSR( LogCalcRoutine, 4, FIT704.value, FIT704.valid, FIT704.log, 55);  //FIT704 - Membrane tank 4 permeate flow
   JSR( LogCalcRoutine, 4, LIT6101.value, LIT6101.valid, LIT6101.log, 56);  //LIT6101 - Coagulant tank level
   JSR( LogCalcRoutine, 4, LIT6102.value, LIT6102.valid, LIT6102.log, 57);  //LIT6102 - Caustic tank level
   JSR( LogMotorRoutine, 2, P802.run_sts, 58 );  //P802 - CIP pump 2
   JSR( LogCalcRoutine, 4, FIT801.value, FIT801.valid, FIT801.log, 59);  //FIT801 - CIP flow
   JSR( LogMotorRoutine, 2, P7951.run_sts, 60 );  //P7951 - Screen building sump pump
   
   
   (* keep track of the last date for the end of the hour *)
   COP(date_time_current,date_time_previous,1);
   
   report_row_daily := report_row;
   
   (* flag that powerup is done *)
   report_pwrup_done := 1;
   
END_ROUTINE
END_PROGRAM

PROGRAM ReportDaily   (* main routine DailyReport *)
// For Displaying Daily Report Data
VAR
   AnyDay : BOOL := 1;
   DATA_RTN_AVG_CALC : REAL := 0.35393435;
   DATA_RTN_MAX_CALC : REAL := 1.0;
   DATA_RTN_MIN_CALC : REAL;
   DATA_RTN_TIME_CALC : REAL := 20298.254;
   DATA_RTN_TOTAL_CALC : REAL := 7184.249;
   DataIndex : INT := 9;
   DayIndex : INT := 7;
   DaysAgo : INT := 6;
   DECIMAL_MULT : DINT;
   DECIMALS : INT := 100;
   HourstoReturn : INT;
   Index : INT := 7;
   INPUTVAL : REAL := 1.9956248;
   INTVAL : DINT := 200;
   Log_Index : INT := 1;
   OUTPUTVAL : REAL := 2.0;
   report_row : INT := 10;
   report_row_qty : INT := 200;
   Retrieve_Count : INT := 6;
   Retrieve_Index : INT := 10;
   Retrieve_Index_Stepper : INT := 7;
   Retrieve_Index_Temp : INT := 34;
   Step_Qty : INT := 24;
   StepIndex : INT := 201;
   SUMMARY_Index_Last : INT := 1;
   Summary_Last_Minute : INT := 13;
   summary_tag_qty : INT := 100;
END_VAR

ROUTINE DailyReport   (* structured text *)
   
END_ROUTINE
END_PROGRAM
